{attribute 'qualified_only'}
{attribute 'strict'}
TYPE ENUM_FirstPass :
(
	Left := 1,
	Right:=0//default
);
END_TYPE

(* stored: Version 1.1.0.1, ProductVersion 3.1.4024.2
   DUT ENUM_FirstPass: Id {b9434211-3471-4ed9-8ca5-3f058be1e857} *)
